RoboDK station: boxes_cells_shelves.rdk

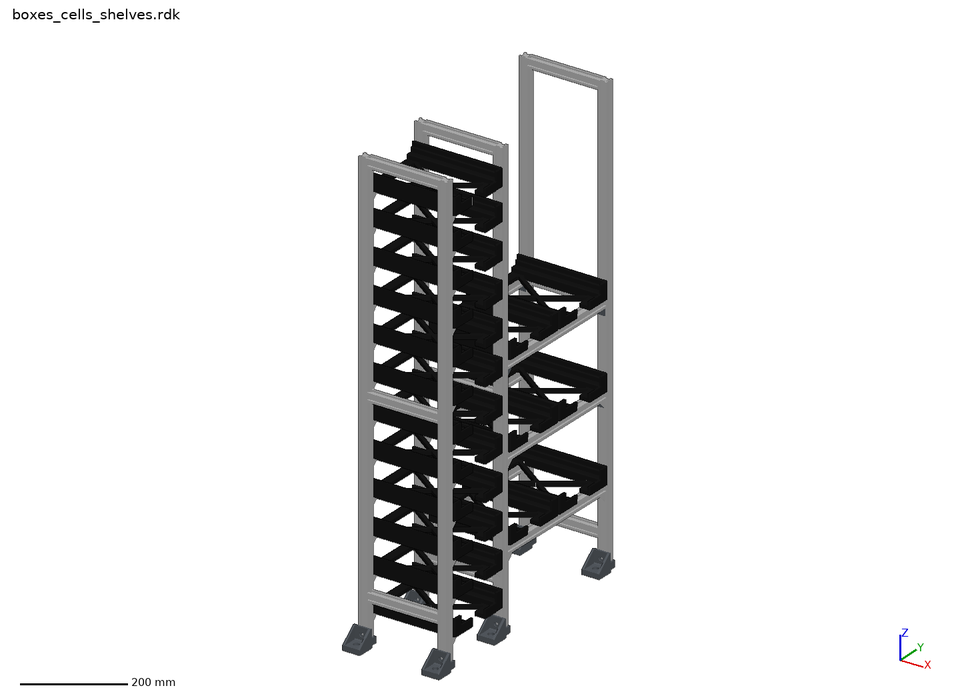
[picture v0: the station drawn from its stored meshes, robots at their saved joint values, targets as dots, program paths as lines]
Station boxes_celss_shelf (saved by RoboDK 5.9.0). Poses are relative to the parent item; angles as X-Y-Z fixed-axis rotations.
  - object boxes_cells_shelf at (0, 0, 0) mm, size 220.1 x 580.5 x 1012 mm, geometry from boxes_cells_shelf.stl
